// TwinCAT 3 PLC project Untitled1
// ProgramVersion: 3.1.4024.0
// libraries:
//   Tc2_Standard, * (Beckhoff Automation GmbH)
//   Tc2_System, * (Beckhoff Automation GmbH)
//   Tc3_Module, * (Beckhoff Automation GmbH)
// project tree:
//   / PlcTask.TcTTO
//   POUs/ MAIN.TcPOU, ST80a.TcPOU, sT80b.TcPOU, ST80c.TcPOU
// real-time tasks:
//   TASK PlcTask: cycle T#10ms, priority 20, ADS port 350

CONFIGURATION Untitled1
    RESOURCE PLC ON TwinCAT3
        TASK PlcTask(INTERVAL := T#10ms, PRIORITY := 20);
        PROGRAM MAIN WITH PlcTask : MAIN;
    END_RESOURCE
END_CONFIGURATION

// ---- POUs/MAIN.TcPOU
PROGRAM MAIN
VAR
	_ST80a		: ST80a;
	_ST80b		: sT80b; 
	_ST80c		: ST80c; 
END_VAR

_ST80a._Ready();

END_PROGRAM

// ---- POUs/ST80a.TcPOU
FUNCTION_BLOCK ST80a
VAR
	_promenlivaIvana	: BOOL;
	_test : BOOL;
	_ivana : BOOL; 
END_VAR

METHOD  _Ready 
VAR_INPUT
END_VAR
_test:= TRUE; 
_promenlivaIvana:= TRUE;
END_METHOD

END_FUNCTION_BLOCK

// ---- POUs/sT80b.TcPOU
FUNCTION_BLOCK sT80b
VAR
	_promenlivataNaFilip : BOOL;
	_test : BOOL; 
END_VAR

METHOD  _test
VAR_INPUT
END_VAR
_promenlivataNaFilip:= TRUE;
_test:= FALSE;
END_METHOD

END_FUNCTION_BLOCK

// ---- POUs/ST80c.TcPOU
FUNCTION_BLOCK ST80c
VAR
	_promenlivaNova		: BOOL;
	_ivana : INT;
	_test : BOOL;
END_VAR

METHOD _test 
VAR_INPUT
END_VAR
IF _test THEN 
	_ivana:= 5;
ELSE 
_ivana:= 3; 
END_IF
END_METHOD

END_FUNCTION_BLOCK
